RESOURCE_TYPE _Core002
  (* Standard: 61499-2 *)
  (* Version 0.1, 2017-00-01, hpea485, UOA *)
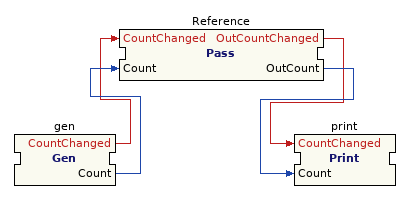
  FBS
    print : Print;
    gen : Gen;
    Reference : Pass;
  END_FBS
  EVENT_CONNECTIONS
    gen.CountChanged TO Reference.CountChanged;
    Reference.OutCountChanged TO print.CountChanged;
  END_CONNECTIONS
  DATA_CONNECTIONS
    gen.Count TO Reference.Count;
    Reference.OutCount TO print.Count;
  END_CONNECTIONS
END_RESOURCE_TYPE
